# EPICS IOC start-up script: iocsh/ethercatmcAnalogOutputReadback.iocsh
ethercatmcCreateAsynParam $(MOTOR_PORT) $(ASYNPARAMNAME)      Float64
ethercatmcCreateAsynParam $(MOTOR_PORT) $(ASYNPARAMNAME)_DESC Octet

dbLoadRecords("ethercatmcAnalogOutputReadback.template", "P=$(P), R=$(R), MOTOR_PORT=$(MOTOR_PORT), CHNO=$(CHNO), ASYNPARAMNAME=$(ASYNPARAMNAME), PREC=$(PREC), DESC=$(DESC), EGU=$(EGU)")
